# EPICS StreamDevice protocol: cm/Db/keithley3706A-pt100.proto
Terminator = LF;
ExtraInput=Ignore;
LockTimeout=9900;

@replytimeout {
    	exec "echo \"reply timeout\""
}
@writetimeout {
    	exec "echo \"write timeout\""
}
@readtimeout {
    	exec "echo \"read timeout\""
}

getId {
        out "*idn?";
        in "KEITHLEY INSTRUMENTS INC.,%#s";
	@init { out "*idn?"; in "KEITHLEY INSTRUMENTS INC.,%#s"; }
}

getUnits {
        out "print(dmm.units)";
        in "%d";
}

getfunc {
        out "print(dmm.func)";
        in "%s";
}

getMeasurement {
        out "channel.close(\"\$10\$2,\$10\$3,\$1911,\$1922\")";
	wait 50;
	out "print(dmm.measure())";
        in "%g";
        out "channel.open(\"allslots\")";
}

#getConnNodes { separator = " ";
#        out "R rci";
#        in "R rci %d";
#   	@init { out "R rci"; in "R rci %d"; }
#}

getRFdataSelf { separator = " ";
        out "R rsd";
        in "R rsd %*d: %d";
}

## Write Only commands

doInit1 {
    out "dmm.func=dmm.FOUR_WIRE_OHMS dmm.autorange=1 dmm.autozero=dmmON";
#    @init {out "dmm.func=dmm.FOUR_WIRE_OHMS dmm.autorange=1 dmm.autozero=dmmON";}
}

doInit2 {
    out "dmm.offsetcompensation=0 dmm.drycircuit=1";
#    @init {out "dmm.offsetcompensation=0 dmm.drycircuit=1";}
}

doInit3 {
    out "dmm.func=dmm.TEMPERATURE dmm.autorange=1 dmm.autozero=dmmON";
    @init {out "dmm.func=dmm.TEMPERATURE dmm.autorange=1 dmm.autozero=dmmON";}
}
doInit4 {
    out "dmm.transducer=dmm.TEMP_FOURRTD dmm.fourrtd=dmm.RTD_PT100 dmm.units=dmm.UNITS_KELVIN dmm.offsetcompensation=0 dmm.drycircuit=1";
    @init {out "dmm.transducer=dmm.TEMP_FOURRTD dmm.fourrtd=dmm.RTD_PT100 dmm.units=dmm.UNITS_KELVIN dmm.offsetcompensation=0 dmm.drycircuit=1";}
}

reset {
    out "*RST";
}

# Connect a stringout record to this to get
# a generic command interface.
# After processing finishes, the record contains the reply.
debug {
ExtraInput = Ignore;
out "%s"; in "%#s;"
}

debugin {
in "%#s"
}
